Fanuc KAREL source: kt00404.KL

-- PROVISIONAL review KL for V1013-1; original PC SHA256 c6642e90f5cfff8ffe9feb94995a311a075d07c25460a2498423450924b1d2ee
-- Incomplete behavior may be omitted. Consult companion uncertainty JSON. Do not deploy.
PROGRAM KT00404
%NOLOCKGROUP
VAR
  I1 : INTEGER
  OUT : BOOLEAN
-- UNRESOLVED_DECL H2 type=002017
BEGIN
  -- UNRESOLVED_PC offsets 5-16; opcodes 2E,23
  -- UNRESOLVED_PC offsets 21-35; opcodes 2E,22,9D,33,B4
  -- UNRESOLVED_PC offsets 40-62; opcodes 21,22,9D,33,B3,5B,23
  -- UNRESOLVED_PC offsets 67-71; opcodes 7F
END KT00404
